{attribute 'linkalways'} 
{attribute 'no_explicit_call' := 'This FB is a CLASS and must be accessed using methods or properties'}
{attribute 'enable_dynamic_creation'}
FUNCTION_BLOCK _ETcVnMorphologicalOperator EXTENDS EnumDatatypeBase
VAR
	localData : ETcVnMorphologicalOperator;
	activeData : REFERENCE TO ETcVnMorphologicalOperator;
	enumBaseDatatype : _DINT(localData);
END_VAR

METHOD PRIVATE AddLocalEnumeration
VAR_INPUT
	Enumeration : T_MAXSTRING;
	Value : ETcVnMorphologicalOperator;
END_VAR
AddEnumeration(Enumeration, Value);
END_METHOD

PROPERTY PUBLIC Address : PVOID
GET
Address := ADR(activeData);
END_GET
END_PROPERTY

METHOD PUBLIC ClearReference
VAR_INPUT
END_VAR
activeData REF= localData;
SetBaseDatatypeReference();
END_METHOD

METHOD PUBLIC Clone : I_Datatype
VAR
    pClone : POINTER TO _ETcVnMorphologicalOperator;
END_VAR
pClone := __NEW(_ETcVnMorphologicalOperator(InitialValue := Value));
Clone := pClone^;
END_METHOD

METHOD FB_init : BOOL
VAR_INPUT
	bInitRetains : BOOL; // if TRUE, the retain variables are initialized (warm start / cold start)
	bInCopyCode : BOOL;  // if TRUE, the instance afterwards gets moved into the copy code (online change)
	InitialValue : ETcVnMorphologicalOperator;
END_VAR
localData := InitialValue;
AddBaseDatatype(enumBaseDatatype);
ClearReference();

AddLocalEnumeration('TCVN_MO_EROSION', ETcVnMorphologicalOperator.TCVN_MO_EROSION);
AddLocalEnumeration('TCVN_MO_DILATION', ETcVnMorphologicalOperator.TCVN_MO_DILATION);
AddLocalEnumeration('TCVN_MO_OPENING', ETcVnMorphologicalOperator.TCVN_MO_OPENING);
AddLocalEnumeration('TCVN_MO_CLOSING', ETcVnMorphologicalOperator.TCVN_MO_CLOSING);
AddLocalEnumeration('TCVN_MO_GRADIENT', ETcVnMorphologicalOperator.TCVN_MO_GRADIENT);
AddLocalEnumeration('TCVN_MO_WHITE_TOPHAT', .TCVN_MO_WHITE_TOPHAT);
AddLocalEnumeration('TCVN_MO_BLACK_TOPHAT', ETcVnMorphologicalOperator.TCVN_MO_BLACK_TOPHAT);
AddLocalEnumeration('TCVN_MO_OPENING_BY_RECONSTRUCTION', ETcVnMorphologicalOperator.TCVN_MO_OPENING_BY_RECONSTRUCTION);
AddLocalEnumeration('TCVN_MO_CLOSING_BY_RECONSTRUCTION', ETcVnMorphologicalOperator.TCVN_MO_CLOSING_BY_RECONSTRUCTION);
AddLocalEnumeration('TCVN_MO_WHITE_TOPHAT_BY_RECONSTRUCTION', ETcVnMorphologicalOperator.TCVN_MO_WHITE_TOPHAT_BY_RECONSTRUCTION);
AddLocalEnumeration('TCVN_MO_BLACK_TOPHAT_BY_RECONSTRUCTION', ETcVnMorphologicalOperator.TCVN_MO_BLACK_TOPHAT_BY_RECONSTRUCTION);
END_METHOD

PROPERTY PUBLIC Identifier : T_MAXSTRING
GET
Identifier := 'ETcVnMorphologicalOperator';
END_GET
END_PROPERTY

METHOD IsEnumeratorValueEqual : BOOL
VAR_INPUT
	Enumerator : I_KeyValueForwardEnumerator;
END_VAR
VAR
	storedValue : ETcVnMorphologicalOperator;
END_VAR
IF NOT Enumerator.TryGet(storedValue) THEN
	RETURN;
END_IF

IsEnumeratorValueEqual := storedValue = activeData;
END_METHOD

METHOD PUBLIC MakeReferenceTo
VAR_INPUT
	ReferenceTarget : REFERENCE TO ETcVnMorphologicalOperator;
END_VAR
activeData REF= ReferenceTarget;
SetBaseDatatypeReference();
END_METHOD

METHOD PROTECTED SetBaseDatatypeReference
VAR_INPUT
END_VAR
enumBaseDatatype.MakeReferenceTo(activeData);
END_METHOD

PROPERTY PUBLIC Size : UDINT
GET
Size := SIZEOF(activeData);
END_GET
END_PROPERTY

METHOD TryMakeReferenceTo : BOOL
VAR_INPUT
	Target : I_Datatype;
END_VAR
VAR
	targetAsEnum : I_EnumDatatype;
	pTargetData : POINTER TO ETcVnMorphologicalOperator;
END_VAR
IF NOT Target.TryResolveAsEnumDatatype(targetAsEnum) THEN
	RETURN;
END_IF

IF targetAsEnum.Identifier <> Identifier THEN
	RETURN;
END_IF

pTargetData := Target.Address;
activeData REF= pTargetData^;
SetBaseDatatypeReference();
TryMakeReferenceTo := TRUE;
END_METHOD

PROPERTY PUBLIC Value : ETcVnMorphologicalOperator
GET
Value := activeData;
END_GET
SET
activeData := Value;
END_SET
END_PROPERTY

END_FUNCTION_BLOCK

(* stored: Version 1.1.0.1, ProductVersion 3.1.4024.12
   POU _ETcVnMorphologicalOperator: Id {4ab1e0f4-6c56-09a8-21ee-344468a56821}, SpecialFunc None
   Folder Constructor: Id {1ec0e912-4d71-0601-0dea-d94b281e3869}
   Folder Private: Id {0a6917d4-3746-09ed-3837-a0a287b50a76}
   Folder Protected: Id {f0d60536-b5af-00c6-0ddb-b736ff246915}
   Method AddLocalEnumeration: Id {a5338993-670c-0145-098d-4d5e6675a300}
   Property Address: Id {08e169dc-3ff8-0211-381b-2666c1536ad9}
   Get Get: Id {ee5a3019-0cd7-003b-38cb-181c2b92cc40}
   Method ClearReference: Id {ac9db173-6b6e-0fe2-070d-48517a2b41b9}
   Method Clone: Id {47c15e73-5191-0991-3620-b30cec27d17a}
   Method FB_init: Id {f40362a7-5531-0016-0ced-db909a4e8d3e}
   Property Identifier: Id {df116bcc-cc2b-0160-3720-89be68cc529b}
   Get Get: Id {a804f63b-b517-0dc3-1ad8-31255298e695}
   Method IsEnumeratorValueEqual: Id {b778d932-d482-0010-3ce3-9fc8b7df8bfd}
   Method MakeReferenceTo: Id {284b87fd-6e7e-0319-3d33-92e6391868e2}
   Method SetBaseDatatypeReference: Id {8f2e7931-2938-0180-1772-99d5ce48016a}
   Property Size: Id {34dc30cd-1e8d-07d7-0cb6-b1250146d267}
   Get Get: Id {316ca919-7d6f-0d57-1db7-b51bcf558485}
   Method TryMakeReferenceTo: Id {bca86c23-63e5-090d-384c-33f9b35d57da}
   Property Value: Id {8d30fc7a-5928-03ce-1f16-a960ff54abaf}
   Get Get: Id {b25e9e74-6a14-00cd-20ff-fc4773d5912d}
   Set Set: Id {a3a741b4-0d9d-023c-1469-f80cf2de6e7d} *)
